PROGRAM Background_GPS

VAR
	RxBuffer	:ComBuffer;
	TxBuffer	:ComBuffer;
	
	fbLineCtrlAds	: SerialLineControlADS;
	bAdsError		: BOOL;
	nAdsErrorID		: UDINT;
	bConnect		: BOOL := TRUE;
	sNetID			: T_amsNetId;
	stSerialCfg		: ComSerialConfig;
	Port			: BOOL;
END_VAR

stSerialCfg.Baudrate := 4800;
stSerialCfg.ComPort := 3;
stSerialCfg.DataBits := 8;
stSerialCfg.Parity := PARITY_NONE;
stSerialCfg.StopBits := STOPBITS_ONE;

fbLineCtrlAds(
	Connect 	:= bConnect,
	SerialCfg	:= stSerialCfg,
	NetId		:= sNetId,
	Timeout		:= T#5s,
	TxBuffer	:= TxBuffer,
	RxBuffer	:= RxBuffer,
	Busy		:= ,
	Error		=> bAdsError,
	ErrorID		=> nAdsErrorID,
	PortOpened	=> Port
);

END_PROGRAM

(* stored: Version 1.1.0.1, ProductVersion 3.1.4024.6
   POU Background_GPS: Id {d21b8d5b-1fe8-418c-aa61-d85ef3e640c3}, SpecialFunc None *)
